// TIA Portal V17 export
// export: Created 2024-09-15T12:30:22.4533908Z, ExportSetting WithDefaults, DisplayName Totally Integrated Automation Portal, DisplayVersion V17, DisplayName TIA Portal Openness, DisplayVersion V17, DisplayName TIA Portal Version Control Interface, DisplayVersion V17, DisplayName STEP 7 Professional, DisplayVersion V17, DisplayName STEP 7 Safety, DisplayVersion V17, DisplayName WinCC Professional, DisplayVersion V17
VAR_GLOBAL   // PLC tag table "Global"
   IX_Set_Park_Position AT %I4.7 : Bool;
END_VAR
VAR_GLOBAL CONSTANT   // user constants
   Ci_Queue_Length : Int := 6;
END_VAR
